TYPE ST_SystemTime :
STRUCT
	AutoSyncToGPS	:	BOOL;
	ManualSync		:	BOOL;
	ManSyncValue	:	DT;
END_STRUCT
END_TYPE

(* stored: Version 1.1.0.1, ProductVersion 3.1.4026.18
   DUT ST_SystemTime: Id {3f3715fe-96e9-4820-bd99-d09c69fbd86f} *)
